FUNCTION_BLOCK TEST_GTN (* Test GT functions of numerical values *)
  (* Standard: IEC 61499-1 *)
  (* Version 0.0, 2006-09-11, JHC, Holobloc Inc *)
  (* Compiler header: package fb.rt.test; *)
  (* Compiler classdef: SimpleFB *)
  (* Compiler Java Sun JDK 1.5.0 *)
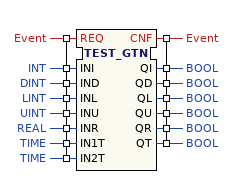
  EVENT_INPUT
    REQ WITH INI, INL, INU, IND, INR, IN1T, IN2T;
  END_EVENT
  EVENT_OUTPUT
    CNF WITH QI, QD, QL, QU, QR, QT;
  END_EVENT
  VAR_INPUT
    INI : INT;
    IND : DINT;
    INL : LINT;
    INU : UINT;
    INR : REAL;
    IN1T : TIME;
    IN2T : TIME;
  END_VAR
  VAR_OUTPUT
    QI : BOOL;
    QD : BOOL;
    QL : BOOL;
    QU : BOOL;
    QR : BOOL;
    QT : BOOL;
  END_VAR
  ALGORITHM REQ IN FBD:
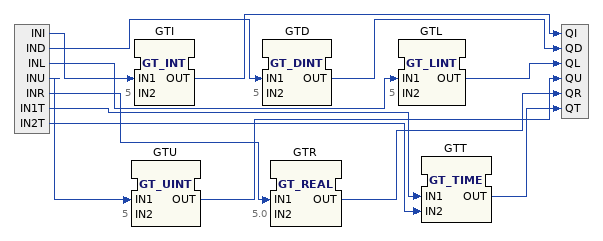
    FBS
      GTI : GT_INT(IN2 := 5);
      GTD : GT_DINT(IN2 := 5);
      GTL : GT_LINT(IN2 := 5);
      GTU : GT_UINT(IN2 := 5);
      GTR : GT_REAL(IN2 := 5.0);
      GTT : GT_TIME;
    END_FBS
    DATA_CONNECTIONS
      INI TO GTI.IN1;
      IND TO GTD.IN1;
      INL TO GTL.IN1;
      INU TO GTU.IN1;
      INR TO GTR.IN1;
      GTI.OUT TO QI;
      GTD.OUT TO QD;
      GTL.OUT TO QL;
      GTU.OUT TO QU;
      GTR.OUT TO QR;
      GTT.OUT TO QT;
      IN1T TO GTT.IN1;
      IN2T TO GTT.IN2;
    END_CONNECTIONS
  END_ALGORITHM
END_FUNCTION_BLOCK
